FUNCTION_BLOCK FB85
TITLE = 'process'
AUTHOR : CB

VAR
	process_F1 : FB79;
	process_F2 : FB81;
	process_F3 : FB83;
END_VAR


BEGIN


NETWORK
TITLE =
//
//	process/MGT1PROC
CALL FC77 (combE := 1);
CALL FB77,	DB77;
CALL FC77 (combE := 0);



NETWORK
TITLE =
//
//	process/process_F1
CALL #process_F1;



NETWORK
TITLE =
//
//	process/process_F2
CALL #process_F2;



NETWORK
TITLE =
//
//	process/process_F3
CALL #process_F3;




END_FUNCTION_BLOCK
